TYPE ST_Encoder_Config :
STRUCT
	bIsIntegrator   		: BOOL := FALSE;  //Integrate input value
	fNumerator 	  			: REAL := 0.0001; //[unit/INC]
	fDenominator  			: REAL := 1.0; 	// Scaling
	fModulo 	  			: REAL := 0; // Modulo [unit]; If 0, will be ignored
	fGearFactor  			: REAL := 1.0;
	bInvertEncoderDirection : BOOL;
END_STRUCT
END_TYPE

(* stored: Version 1.1.0.1, ProductVersion 3.1.4024.12
   DUT ST_Encoder_Config: Id {b88c6e33-7612-0ba9-3961-d0110e3c5c1f} *)
